TEXTLIST SafetyStatusList
  0 = 'SafetyStateNormal'
  1 = 'SafetyStateWarning'
  2 = 'SafetyStateEmergency'
  3 = 'SafetyStateFault'
  4 = 'SafetyStateRecovery'
   = ''
END_TEXTLIST

(* stored: Version 1.1.0.1, ProductVersion 3.1.4024.12
   TextList SafetyStatusList: Id {0ae5047b-f8f6-4069-b777-39919ed2c12d} *)
